{attribute addProperty BoxType "EL2032--0000"}
{attribute addProperty Id "DiagAT %I*ARRAY[0..1] OF Diag_4CD4E3A21620ChannelAT %Q*ARRAY[0..1] OF Channel_7F374EB01620WcStateAT %I*WcState_98A4DF7520.250InfoDataAT %I*InfoData_192954DE1620"}
{attribute addProperty CRC "102408401"}
{attribute addProperty SizeInBites "50"}
{attribute addProperty SizeInBytes "6.25"}
TYPE EL2032_D8352AAE :
STRUCT
	{attribute addProperty Name "Diag"}
	Diag : ARRAY[0..1] OF Diag_4CD4E3A2;
	{attribute addProperty Name "Channel"}
	Channel : ARRAY[0..1] OF Channel_7F374EB0;
	{attribute addProperty Name "WcState"}
	WcState : WcState_98A4DF75;
	{attribute addProperty Name "InfoData"}
	InfoData : InfoData_192954DE;
END_STRUCT
END_TYPE

(* stored: Version 1.2.0.0, ProductVersion 3.1.4024.9
   DUT EL2032_D8352AAE: Id {2ce9dcee-419f-4e8b-9e42-52aed8d7d928} *)
